RoboDK station: lab3_Restrepo&Penagos.rdk

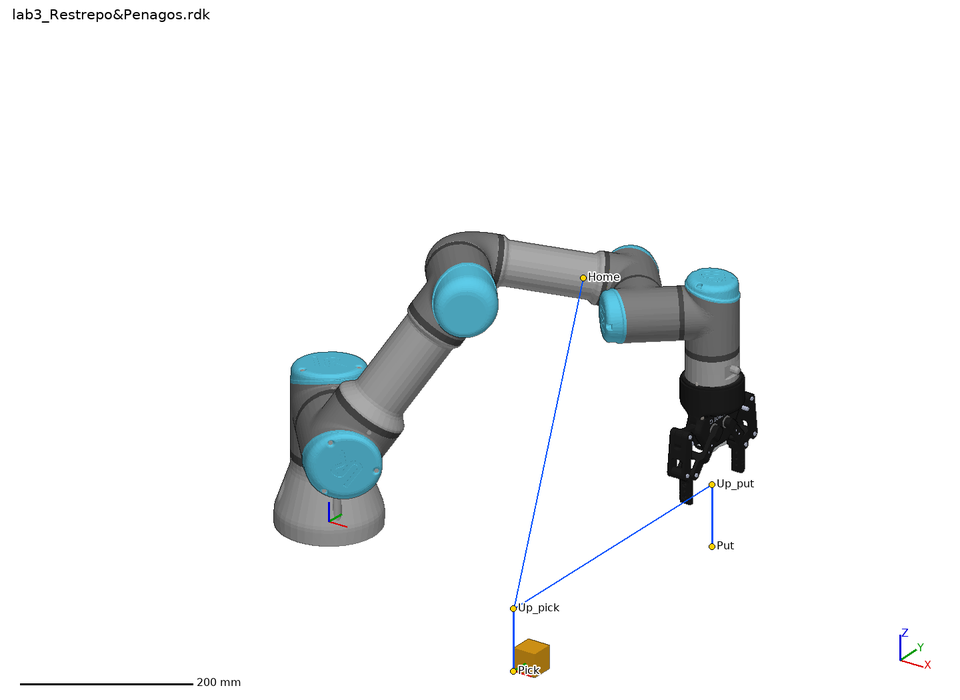
[picture v0: the station drawn from its stored meshes, robots at their saved joint values, targets as dots, program paths as lines]
Station lab3_Restrepo&Penagos (saved by RoboDK 5.6.0). Poses are relative to the parent item; angles as X-Y-Z fixed-axis rotations.
  - frame UR3 Base at (0, 0, 0) mm
    - robot UR3: 6 axes, payload 3 kg, reach 500 mm, repeatability 0.1 mm, weight 11 kg
        modified DH rows (alpha deg, a mm, theta deg, d mm): 0, 0, 0, 151.9; 90, 0, 180, 0; 0, 243.65, 0, 0; 0, 213, 0, 110.4; -90, 0, 0, 83.4; 90, 0, 180, 82.4
        joint limits [-360, -360, -360, -360, -360, -360] to [360, 360, 360, 360, 360, 360]; home [0, -90, -90, 0, 90, 0]; saved at [40.856, -125.72, -67.12, -77.147, 90.001, 40.856]
      - tool RobotiQ 2F-85 Gripper (Open), TCP at (0, 0, 140) mm, size 147.4 x 75 x 146.8 mm
      - tool RobotiQ 2F-85 Gripper (Closed), TCP at (0, 0, 130) mm, size 134.4 x 75 x 157.6 mm
  - frame Frame 2 at (400, -200, 0) mm
    - target Home (Cartesian target) at (35.4, 89.6, 478.95) mm, rotated rx -90 ry 0 rz -90 deg; joints [0, -90, -90, 0, 90, 0] of UR3
    - target Pick (Cartesian target) at (0, 0, 0) mm, rotated rx -179.99 ry 0.01 rz -90 deg; joints [-12.279, -133.005, -77.365, -59.623, 90.011, -12.279] of UR3
    - target Up_pick (Cartesian target) at (0, 0, 80) mm, rotated rx -179.99 ry 0.01 rz -90 deg; joints [-12.279, -125.728, -67.104, -77.161, 90.011, -12.279] of UR3
    - target Up_put (Cartesian target) at (0, 400, 80) mm, rotated rx -179.99 ry 0.01 rz -90 deg; joints [40.856, -125.72, -67.12, -77.147, 90.001, 40.856] of UR3
    - target Put (Cartesian target) at (0, 400, 0) mm, rotated rx -179.99 ry 0.01 rz -90 deg; joints [40.856, -132.999, -77.379, -59.609, 90.001, 40.856] of UR3
    - object Box at (0, 0, 0) mm, size 30 x 30 x 30 mm, geometry from Cube-100mm.sld
  - program Prog1 (16 instructions, listed below)
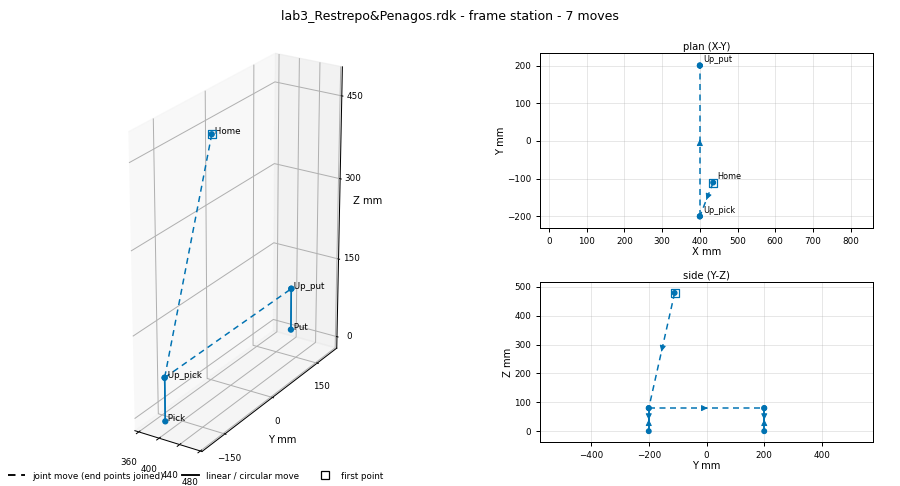
[picture p0: tool path of lab3_Restrepo&Penagos.rdk in frame station, 7 of 7 moves have a stored position in this frame; points joined in program order, loops and branches not executed]

--- program Prog1 (robot UR3) ---
  Set Ref.: Frame 2
  Set Tool: RobotiQ 2F-85 Gripper (Open)
  MoveJ (Home)
  MoveJ (Up_pick)
  MoveL (Pick)
  Ocultar RobotiQ 2F-85 Gripper (Open)
  Mostrar RobotiQ 2F-85 Gripper (Closed)
  Adjuntar a RobotiQ 2F-85 Gripper (Open)
  MoveL (Up_pick)
  MoveJ (Up_put)
  MoveL (Put)
  Ocultar RobotiQ 2F-85 Gripper (Closed)
  Mostrar RobotiQ 2F-85 Gripper (Open)
  Separar de RobotiQ 2F-85 Gripper (Open)
  MoveL (Up_put)
  Reemplazar Box
